// TIA Portal project "FactoryIO_Template" (V17)

(* hardware
DEVICE "S71500/ET200MP-Station_1"  S7-1500 station
   slot 0: "Profilschiene_0"  6ES7 590-1***0-0AA0
   slot 1: "PLC_1"  CPU 1511-1 PN  6ES7 511-1AK00-0AB0  V1.8
   slot 2: "AI 8xU/I/RTD/TC ST_1"  AI 8xU/I/RTD/TC ST  6ES7 531-7KF00-0AB0  V2.0
   slot 3: "AI 8xU/I/RTD/TC ST_2"  AI 8xU/I/RTD/TC ST  6ES7 531-7KF00-0AB0  V2.0
   slot 4: "AI 8xU/I/RTD/TC ST_3"  AI 8xU/I/RTD/TC ST  6ES7 531-7KF00-0AB0  V2.0
   slot 5: "AI 8xU/I/RTD/TC ST_4"  AI 8xU/I/RTD/TC ST  6ES7 531-7KF00-0AB0  V2.0
   slot 6: "DI 16x24VDC BA_1"  DI 16x24VDC BA  6ES7 521-1BH10-0AA0  V1.0
DEVICE "HMI_1"  TP700 Comfort
   slot 0: "HMI_1"  TP700 Comfort  6AV2 124-0GC01-0AX0  17.0.0.0
   slot 1: "HMI_RT_1"  TP700 Comfort  6AV2 124-0GC01-0AX0  17.0.0.0
   slot 5: "HMI_1.IE_CP_1"  PROFINET Interface  17.0.0.0
      slot 1: "PROFINET Interface_1"  PROFINET Interface
         slot 1: "Port_1"  Port
         slot 2: "Port_2"  Port
   slot 7: "HMI_1.MPI/DP_CP_1"  MPI/DP Interface  17.0.0.0
*)

// ===== PLC "PLC_1"  CPU 1511-1 PN =====

VAR_GLOBAL   // PLC tag table "Standard-Variablentabelle"
   "S" AT %E0.0 : Bool;   // capteur de présence du flacon sur le convoyeur 1
   "S21" AT %I0.7 : Bool;   // Convoyeur1
   "FCY" AT %I0.1 : Bool;   // arret urgence
   "DCY" AT %I0.3 : Bool;   // ok button
   "Me_1" AT %M0.0 : Bool;
   "EV" AT %Q0.1 : Bool;
   "S2" AT %I0.2 : Bool;
   "C2" AT %Q0.2 : Bool;
   "Me_2" AT %M0.1 : Bool;
   "C1" AT %Q0.0 : Bool;
   "movingX" AT %I0.5 : Bool;
   "movingZ" AT %I0.6 : Bool;
   "detected" AT %I0.4 : Bool;
   "pickZ" AT %Q0.3 : Bool;
   "pickX" AT %Q0.4 : Bool;
   "grab" AT %Q0.5 : Bool;
   "Tag_1" AT %M0.2 : Bool;
   "Tag_2" AT %M0.3 : Bool;
   "Tag_3" AT %M0.4 : Bool;
   "Tag_4" AT %M0.5 : Bool;
   "Tag_5" AT %M0.7 : Bool;
   "Tag_6" AT %M1.0 : Bool;
   "Tag_7" AT %M1.1 : Bool;
   "sd" AT %I1.0 : Bool;
   "cb" AT %Q0.6 : Bool;
   "Tag_8" AT %M1.2 : Bool;
   "Tag_9" AT %M1.3 : Bool;
   "Tag_10" AT %M1.4 : Bool;
   "Tag_11" AT %M1.5 : Bool;
   "C3" AT %Q0.7 : Bool;
   "AU" AT %I1.1 : Bool;
   "C4" AT %Q1.0 : Bool;
   "C6" AT %Q1.2 : Bool;
   "S3" AT %I1.2 : Bool;
   "C5" AT %Q1.1 : Bool;
   "S45" AT %I1.3 : Bool;
   "S5" AT %I1.4 : Bool;
   "Tag_12" AT %M1.6 : Bool;
   "C7" AT %Q1.3 : Bool;
   "S6" AT %I1.5 : Bool;
   "Tag_14" AT %M1.7 : Bool;
   "Tag_13" AT %M2.0 : Bool;
   "Tag_15" AT %M2.1 : Bool;
   "X" AT %QD30 : Real;
   "Z" AT %QD34 : Real;
   "Tag_16" AT %I1.6 : Bool;
   "Tag_17" AT %M2.2 : Bool;
   "Tag_18" AT %Q1.4 : Bool;
   "ZP" AT %ID30 : Real;
   "Tag_19" AT %M2.3 : Bool;
   "SensorZ" AT %I1.7 : Bool;
   "Tag_21" AT %M2.4 : Bool;
   "Tag_20" AT %Q1.5 : Bool;
   "Tag_22" AT %I2.1 : Bool;
   "Tag_23" AT %I2.0 : Bool;
   "Tag_24" AT %M2.5 : Bool;
   "start" AT %I2.2 : Bool;
   "Tag_26" AT %M2.6 : Bool;
   "Tag_27" AT %M2.7 : Bool;
   "C8" AT %Q1.6 : Bool;
   "Tag_30" AT %Q1.7 : Bool;
   "Tag_32" AT %M3.0 : Bool;
   "full" AT %I2.6 : Bool;
   "Tag_33" AT %M3.1 : Bool;
   "low" AT %I2.7 : Bool;
   "Tag_35" AT %Q2.5 : Bool;
   "Tag_36" AT %M3.2 : Bool;
   "discharge" AT %Q2.6 : Bool;
   "SS" AT %I2.3 : Bool;
   "startIHM" AT %I2.4 : Bool;
   "Tag_25" AT %M3.3 : Bool;
   "Tag_28" AT %M3.4 : Bool;
   "Tag_29" AT %M3.5 : Bool;
   "Tag_31" AT %I2.5 : Bool;
   "Tag_34" AT %M3.6 : Bool;
   "Tag_37" AT %MW4 : Int;
   "Tag_38" AT %M4.0 : Bool;
   "cv" AT %MW6 : Int;
   "Tag_39" AT %M4.1 : Bool;
END_VAR

// folder: System blocks/Program resources

DATA_BLOCK "T1"   // DB1
{ S7_Optimized_Access := 'TRUE' }
AUTHOR : Simatic
FAMILY : IEC
NAME : IEC_TMR
VERSION : 1.0
// stored: InstanceOfName IEC_TIMER
"IEC_TIMER"
BEGIN
END_DATA_BLOCK

DATA_BLOCK "T2"   // DB2
{ S7_Optimized_Access := 'TRUE' }
AUTHOR : Simatic
FAMILY : IEC
NAME : IEC_TMR
VERSION : 1.0
// stored: InstanceOfName IEC_TIMER
"IEC_TIMER"
BEGIN
END_DATA_BLOCK

DATA_BLOCK "T3"   // DB3
{ S7_Optimized_Access := 'TRUE' }
AUTHOR : Simatic
FAMILY : IEC
NAME : IEC_TMR
VERSION : 1.0
// stored: InstanceOfName IEC_TIMER
"IEC_TIMER"
BEGIN
END_DATA_BLOCK

DATA_BLOCK "T4"   // DB4
{ S7_Optimized_Access := 'TRUE' }
AUTHOR : Simatic
FAMILY : IEC
NAME : IEC_TMR
VERSION : 1.0
// stored: InstanceOfName IEC_TIMER
"IEC_TIMER"
BEGIN
END_DATA_BLOCK

DATA_BLOCK "com1"   // DB5
{ S7_Optimized_Access := 'TRUE' }
AUTHOR : Simatic
FAMILY : IEC
NAME : CNTR
VERSION : 1.0
// stored: InstanceOfName IEC_COUNTER
"IEC_COUNTER"
BEGIN
END_DATA_BLOCK

// folder: (top level)

FUNCTION "MHJ-PLC-Lab-Function-S71500" : Void   // FC9000, SCL
{ S7_Optimized_Access := 'TRUE' }
VERSION : 0.1
   VAR_TEMP
      Value : Byte;
      ForCounter : Int;
   END_VAR
   VAR CONSTANT
      Value_01_DW : DWord := 16#1223_5486;
      Value_02_DW : DWord := 16#A6C9_D1F5;
   END_VAR
BEGIN

   #Value:=PEEK(area := 16#82,
        dbNumber := 0,
        byteOffset := 511);
   #Value := #Value + 1;

   POKE(area := 16#82,
        dbNumber := 0,
        byteOffset := 511,
        value := #Value);

   POKE(area := 16#82,
        dbNumber := 0,
        byteOffset := 1016,
        value := #Value_01_DW);
   POKE(area := 16#82,
        dbNumber := 0,
        byteOffset := 1020,
        value := #Value_02_DW);

   FOR #ForCounter := 0 TO 63 DO
       #Value:=PEEK(area := 16#1,
            dbNumber := 0,
            byteOffset := #ForCounter);
       POKE(area := 16#81,
            dbNumber := 0,
            byteOffset := #ForCounter,
            value := #Value);
   END_FOR;
   #Value := PEEK(area := 16#1,
                  dbNumber := 0,
                  byteOffset := 512);
   POKE(area := 16#82,
        dbNumber := 0,
        byteOffset := 512,
        value := #Value);
END_FUNCTION

ORGANIZATION_BLOCK "Main"   // OB1, LAD, ProgramCycle
TITLE = "Main Program Sweep (Cycle)"
{ S7_Optimized_Access := 'TRUE' }
VERSION : 0.1
   VAR_INPUT
      Initial_Call : Bool;   // Initial call of this OB
      Remanence : Bool;   // =True, if remanent data are available
   END_VAR
   VAR_TEMP   // added for the SCL form of the ladder/FBD networks
      _w1 : Bool;
      _w2 : Bool;
   END_VAR
BEGIN

REGION Network 1
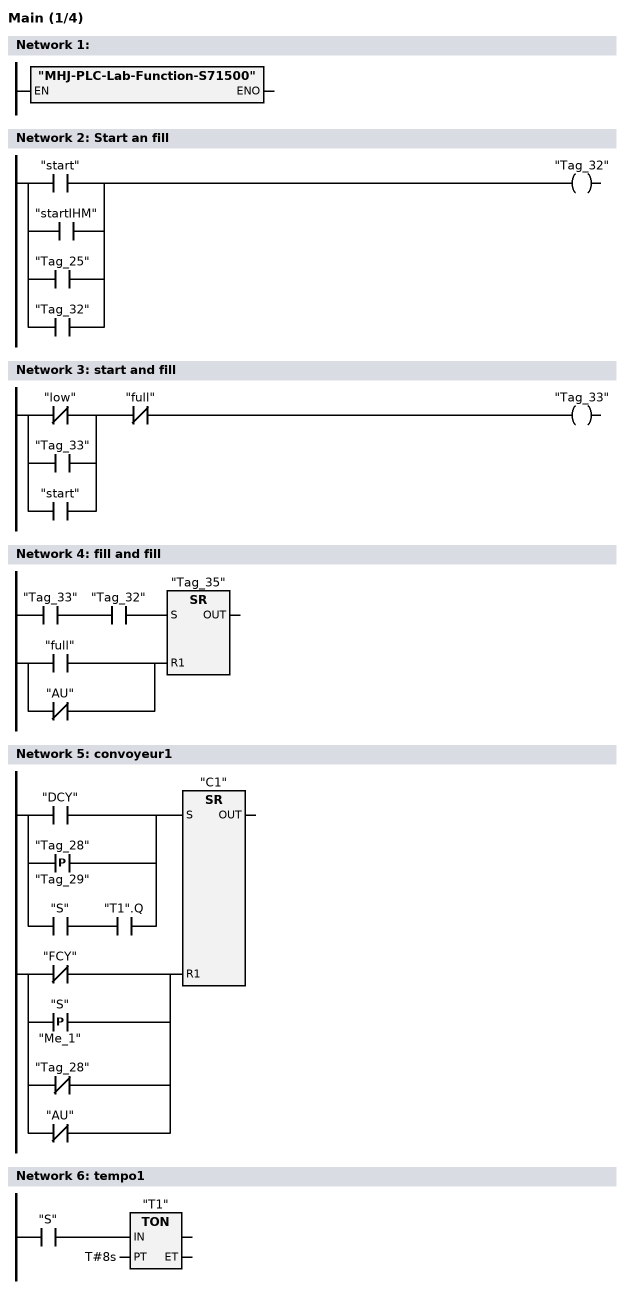
   RUNG wire#powerrail
      "MHJ-PLC-Lab-Function-S71500"()
   END_RUNG
   // the same network as SCL:
   "MHJ-PLC-Lab-Function-S71500"();
END_REGION

REGION Network 2: Start an fill
   RUNG wire#powerrail
      Contact( "start" )
      wire#w1
      Coil( "Tag_32" )
   END_RUNG
   RUNG wire#powerrail
      Contact( "startIHM" )
   END_RUNG wire#w1
   RUNG wire#powerrail
      Contact( "Tag_25" )
   END_RUNG wire#w1
   RUNG wire#powerrail
      Contact( "Tag_32" )
   END_RUNG wire#w1
   // the same network as SCL:
   "Tag_32" := "start" OR "startIHM" OR "Tag_25" OR "Tag_32";
END_REGION

REGION Network 3: start and fill
   RUNG wire#powerrail
      I_Contact( "low" )
      wire#w1
      I_Contact( "full" )
      Coil( "Tag_33" )
   END_RUNG
   RUNG wire#powerrail
      Contact( "Tag_33" )
   END_RUNG wire#w1
   RUNG wire#powerrail
      Contact( "start" )
   END_RUNG wire#w1
   // the same network as SCL:
   "Tag_33" := (NOT "low" OR "Tag_33" OR "start") AND NOT "full";
END_REGION

REGION Network 4: fill and fill
   RUNG wire#powerrail
      Contact( "Tag_33" )
      Contact( "Tag_32" )
      S_SR(operand := "Tag_35", r1 := wire#w1)
   END_RUNG
   RUNG wire#powerrail
      Contact( "full" )
   END_RUNG wire#w1
   RUNG wire#powerrail
      I_Contact( "AU" )
   END_RUNG wire#w1
   // the same network as SCL:
   IF "Tag_33" AND "Tag_32" THEN
       "Tag_35" := TRUE;   // SR flip-flop
   END_IF;
   IF "full" OR NOT "AU" THEN "Tag_35" := FALSE; END_IF;
END_REGION

REGION Network 5: convoyeur1
   RUNG wire#powerrail
      Contact( "DCY" )
      wire#w1
      S_SR(operand := "C1", r1 := wire#w2)
   END_RUNG
   RUNG wire#powerrail
      P_Contact(operand := "Tag_28", bit := "Tag_29")
   END_RUNG wire#w1
   RUNG wire#powerrail
      Contact( "S" )
      Contact( "T1".Q )
   END_RUNG wire#w1
   RUNG wire#powerrail
      I_Contact( "FCY" )
   END_RUNG wire#w2
   RUNG wire#powerrail
      P_Contact(operand := "S", bit := "Me_1")
   END_RUNG wire#w2
   RUNG wire#powerrail
      I_Contact( "Tag_28" )
   END_RUNG wire#w2
   RUNG wire#powerrail
      I_Contact( "AU" )
   END_RUNG wire#w2
   // the same network as SCL:
   #_w1 := "Tag_28" AND NOT "Tag_29";   // rising edge of "Tag_28"
   "Tag_29" := "Tag_28";
   #_w2 := "S" AND NOT "Me_1";   // rising edge of "S"
   "Me_1" := "S";
   IF "DCY" OR #_w1 OR ("S" AND "T1".Q) THEN
       "C1" := TRUE;   // SR flip-flop
   END_IF;
   IF NOT "FCY" OR #_w2 OR NOT "Tag_28" OR NOT "AU" THEN "C1" := FALSE; END_IF;
END_REGION

REGION Network 6: tempo1
   "T1".TON(IN := "S", PT := T#8s);
END_REGION

REGION Network 7: electrovanne
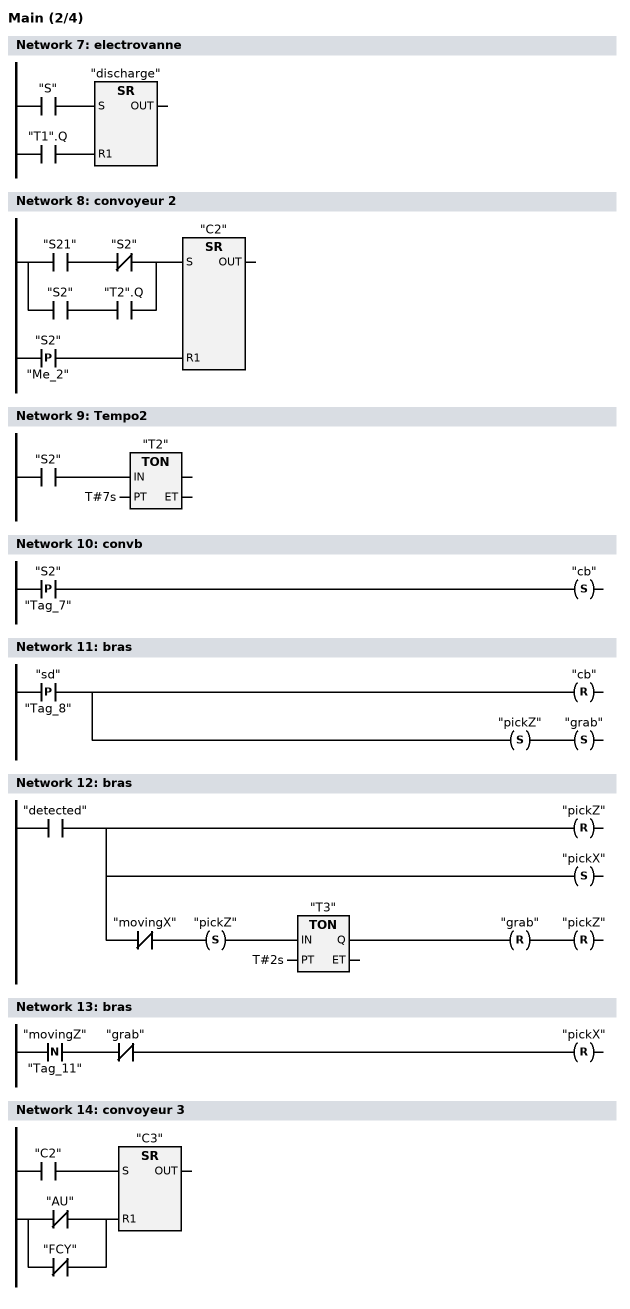
   RUNG wire#powerrail
      Contact( "S" )
      S_SR(operand := "discharge", r1 := wire#w1)
   END_RUNG
   RUNG wire#powerrail
      Contact( "T1".Q )
   END_RUNG wire#w1
   // the same network as SCL:
   IF "S" THEN
       "discharge" := TRUE;   // SR flip-flop
   END_IF;
   IF "T1".Q THEN "discharge" := FALSE; END_IF;
END_REGION

REGION Network 8: convoyeur 2
   RUNG wire#powerrail
      Contact( "S21" )
      I_Contact( "S2" )
      wire#w1
      S_SR(operand := "C2", r1 := wire#w2)
   END_RUNG
   RUNG wire#powerrail
      Contact( "S2" )
      Contact( "T2".Q )
   END_RUNG wire#w1
   RUNG wire#powerrail
      P_Contact(operand := "S2", bit := "Me_2")
   END_RUNG wire#w2
   // the same network as SCL:
   #_w1 := "S2" AND NOT "Me_2";   // rising edge of "S2"
   "Me_2" := "S2";
   IF ("S21" AND NOT "S2") OR ("S2" AND "T2".Q) THEN
       "C2" := TRUE;   // SR flip-flop
   END_IF;
   IF #_w1 THEN "C2" := FALSE; END_IF;
END_REGION

REGION Network 9: Tempo2
   "T2".TON(IN := "S2", PT := T#7s);
END_REGION

REGION Network 10: convb
   RUNG wire#powerrail
      P_Contact(operand := "S2", bit := "Tag_7")
      S_Coil( "cb" )
   END_RUNG
   // the same network as SCL:
   #_w1 := "S2" AND NOT "Tag_7";   // rising edge of "S2"
   "Tag_7" := "S2";
   IF #_w1 THEN "cb" := TRUE; END_IF;
END_REGION

REGION Network 11: bras
   RUNG wire#powerrail
      P_Contact(operand := "sd", bit := "Tag_8")
      wire#w1
      R_Coil( "cb" )
   END_RUNG
   RUNG wire#w1
      S_Coil( "pickZ" )
      S_Coil( "grab" )
   END_RUNG
   // the same network as SCL:
   #_w1 := "sd" AND NOT "Tag_8";   // rising edge of "sd"
   "Tag_8" := "sd";
   IF #_w1 THEN
       "cb" := FALSE;
       "pickZ" := TRUE;
       "grab" := TRUE;
   END_IF;
END_REGION

REGION Network 12: bras
   IF "detected" THEN
       "pickZ" := FALSE;
       "pickX" := TRUE;
   END_IF;
   #_w1 := "detected" AND NOT "movingX";
   IF #_w1 THEN "pickZ" := TRUE; END_IF;
   "T3".TON(IN := #_w1, PT := T#2s);
   IF "T3".Q THEN
       "grab" := FALSE;
       "pickZ" := FALSE;
   END_IF;
END_REGION

REGION Network 13: bras
   RUNG wire#powerrail
      N_Contact(operand := "movingZ", bit := "Tag_11")
      I_Contact( "grab" )
      R_Coil( "pickX" )
   END_RUNG
   // the same network as SCL:
   #_w1 := NOT "movingZ" AND "Tag_11";   // falling edge of "movingZ"
   "Tag_11" := "movingZ";
   IF #_w1 AND NOT "grab" THEN "pickX" := FALSE; END_IF;
END_REGION

REGION Network 14: convoyeur 3
   RUNG wire#powerrail
      Contact( "C2" )
      S_SR(operand := "C3", r1 := wire#w1)
   END_RUNG
   RUNG wire#powerrail
      I_Contact( "AU" )
   END_RUNG wire#w1
   RUNG wire#powerrail
      I_Contact( "FCY" )
   END_RUNG wire#w1
   // the same network as SCL:
   IF "C2" THEN
       "C3" := TRUE;   // SR flip-flop
   END_IF;
   IF NOT "AU" OR NOT "FCY" THEN "C3" := FALSE; END_IF;
END_REGION

REGION Network 15: convoyeur 4
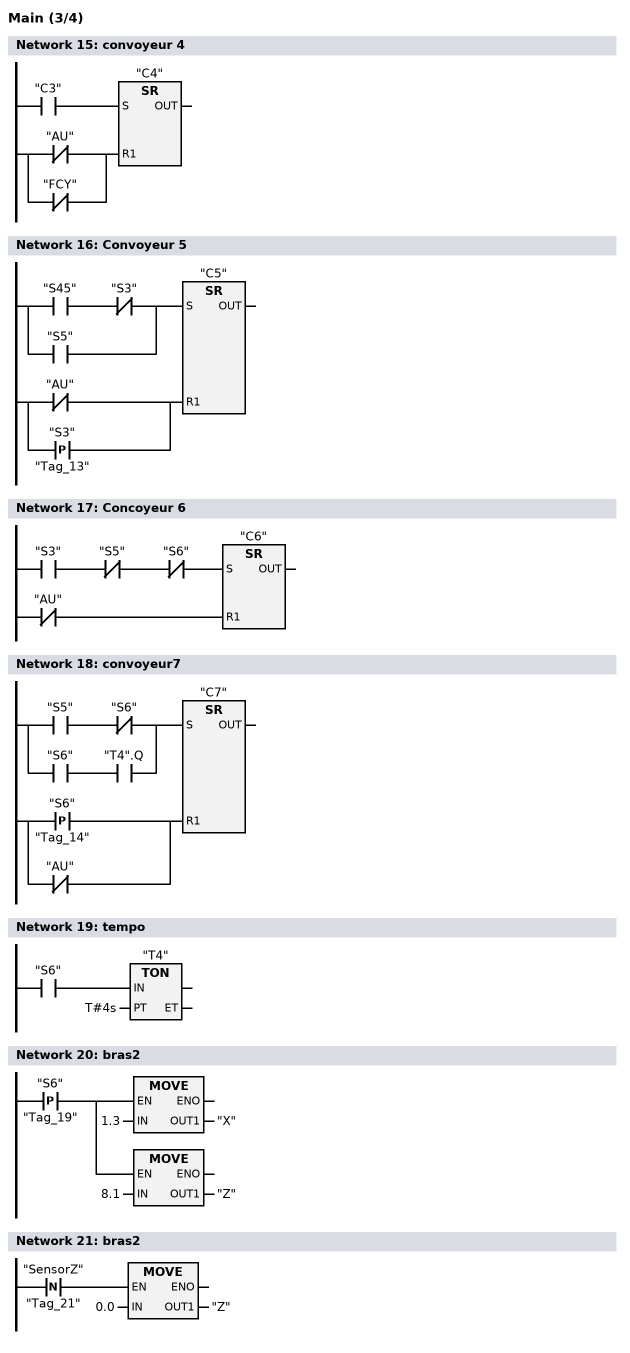
   RUNG wire#powerrail
      Contact( "C3" )
      S_SR(operand := "C4", r1 := wire#w1)
   END_RUNG
   RUNG wire#powerrail
      I_Contact( "AU" )
   END_RUNG wire#w1
   RUNG wire#powerrail
      I_Contact( "FCY" )
   END_RUNG wire#w1
   // the same network as SCL:
   IF "C3" THEN
       "C4" := TRUE;   // SR flip-flop
   END_IF;
   IF NOT "AU" OR NOT "FCY" THEN "C4" := FALSE; END_IF;
END_REGION

REGION Network 16: Convoyeur 5
   RUNG wire#powerrail
      Contact( "S45" )
      I_Contact( "S3" )
      wire#w1
      S_SR(operand := "C5", r1 := wire#w2)
   END_RUNG
   RUNG wire#powerrail
      Contact( "S5" )
   END_RUNG wire#w1
   RUNG wire#powerrail
      I_Contact( "AU" )
   END_RUNG wire#w2
   RUNG wire#powerrail
      P_Contact(operand := "S3", bit := "Tag_13")
   END_RUNG wire#w2
   // the same network as SCL:
   #_w1 := "S3" AND NOT "Tag_13";   // rising edge of "S3"
   "Tag_13" := "S3";
   IF ("S45" AND NOT "S3") OR "S5" THEN
       "C5" := TRUE;   // SR flip-flop
   END_IF;
   IF NOT "AU" OR #_w1 THEN "C5" := FALSE; END_IF;
END_REGION

REGION Network 17: Concoyeur 6
   RUNG wire#powerrail
      Contact( "S3" )
      I_Contact( "S5" )
      I_Contact( "S6" )
      S_SR(operand := "C6", r1 := wire#w1)
   END_RUNG
   RUNG wire#powerrail
      I_Contact( "AU" )
   END_RUNG wire#w1
   // the same network as SCL:
   IF "S3" AND NOT "S5" AND NOT "S6" THEN
       "C6" := TRUE;   // SR flip-flop
   END_IF;
   IF NOT "AU" THEN "C6" := FALSE; END_IF;
END_REGION

REGION Network 18: convoyeur7
   RUNG wire#powerrail
      Contact( "S5" )
      I_Contact( "S6" )
      wire#w1
      S_SR(operand := "C7", r1 := wire#w2)
   END_RUNG
   RUNG wire#powerrail
      Contact( "S6" )
      Contact( "T4".Q )
   END_RUNG wire#w1
   RUNG wire#powerrail
      P_Contact(operand := "S6", bit := "Tag_14")
   END_RUNG wire#w2
   RUNG wire#powerrail
      I_Contact( "AU" )
   END_RUNG wire#w2
   // the same network as SCL:
   #_w1 := "S6" AND NOT "Tag_14";   // rising edge of "S6"
   "Tag_14" := "S6";
   IF ("S5" AND NOT "S6") OR ("S6" AND "T4".Q) THEN
       "C7" := TRUE;   // SR flip-flop
   END_IF;
   IF #_w1 OR NOT "AU" THEN "C7" := FALSE; END_IF;
END_REGION

REGION Network 19: tempo
   "T4".TON(IN := "S6", PT := T#4s);
END_REGION

REGION Network 20: bras2
   RUNG wire#powerrail
      P_Contact(operand := "S6", bit := "Tag_19")
      wire#w1
      Move(in := 1.3, out1 => "X")
   END_RUNG
   RUNG wire#w1
      Move(in := 8.1, out1 => "Z")
   END_RUNG
   // the same network as SCL:
   #_w1 := "S6" AND NOT "Tag_19";   // rising edge of "S6"
   "Tag_19" := "S6";
   IF #_w1 THEN
       "X" := 1.3;
       "Z" := 8.1;
   END_IF;
END_REGION

REGION Network 21: bras2
   RUNG wire#powerrail
      N_Contact(operand := "SensorZ", bit := "Tag_21")
      Move(in := 0.0, out1 => "Z")
   END_RUNG
   // the same network as SCL:
   #_w1 := NOT "SensorZ" AND "Tag_21";   // falling edge of "SensorZ"
   "Tag_21" := "SensorZ";
   IF #_w1 THEN "Z" := 0.0; END_IF;
END_REGION

REGION Network 22: Classification
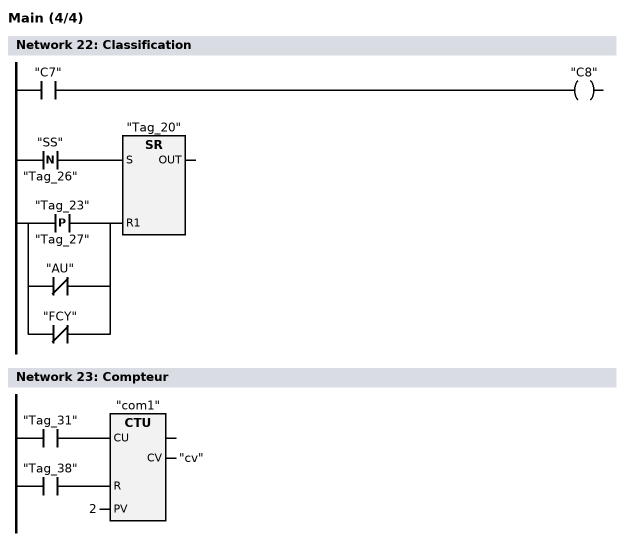
   RUNG wire#powerrail
      Contact( "C7" )
      Coil( "C8" )
   END_RUNG
   RUNG wire#powerrail
      N_Contact(operand := "SS", bit := "Tag_26")
      S_SR(operand := "Tag_20", r1 := wire#w1)
   END_RUNG
   RUNG wire#powerrail
      P_Contact(operand := "Tag_23", bit := "Tag_27")
   END_RUNG wire#w1
   RUNG wire#powerrail
      I_Contact( "AU" )
   END_RUNG wire#w1
   RUNG wire#powerrail
      I_Contact( "FCY" )
   END_RUNG wire#w1
   // the same network as SCL:
   "C8" := "C7";
   #_w1 := NOT "SS" AND "Tag_26";   // falling edge of "SS"
   "Tag_26" := "SS";
   #_w2 := "Tag_23" AND NOT "Tag_27";   // rising edge of "Tag_23"
   "Tag_27" := "Tag_23";
   IF #_w1 THEN
       "Tag_20" := TRUE;   // SR flip-flop
   END_IF;
   IF #_w2 OR NOT "AU" OR NOT "FCY" THEN "Tag_20" := FALSE; END_IF;
END_REGION

REGION Network 23: Compteur
   "com1".CTU(CU := "Tag_31", R := "Tag_38", PV := 2, CV => "cv");
END_REGION
END_ORGANIZATION_BLOCK

(* ===== HMI "HMI_RT_1" =====
system functions are stored by id; their names below are inferred from use
connection "HMI_Connection_1": ETHERNET, S7_1500_OMS

HMI tags "Default tag table"
   "start" : Bool = PLC startIHM AT %I2.4, 1 s
   "AU" : Bool = PLC AU AT %I1.1, 1 s
   "FCY" : Bool = PLC FCY AT %I0.1, 1 s
   "Tag_25" : Bool = PLC Tag_25 AT %M3.3, 1 s
   "Tag_28" : Bool = PLC Tag_28 AT %M3.4, 1 s
   "cv" : Int = PLC cv AT %MW6, 1 s
   "Tag_38" : Bool = PLC Tag_38 AT %M4.0, 1 s

screen "Root screen" 800x420, template "Template_1"
   Button "Button_2" at 291,114 size 132x32; TextOff 'Début cycle'
      on Click: SetBit("Tag_28")
   Button "Button_3" at 527,115 size 96x32; TextOff 'Fin cycle'
      on Click: SetBit("FCY")
   Button "Button_4" at 425,289 size 194x32; TextOff 'Emergency Stop'
      on Click: SetBit("AU")
   Button "Button_5" at 91,114 size 96x32; TextOff 'Start'
      on Click: SetBit("Tag_25")
   IOField "I/O field_2" at 49,289 size 96x32; FormatPattern 999
      ProcessValue <- "cv"
      on Deactivate: ResetBit(N)
   Button "Button_1" at 40,238 size 253x32; TextOff 'Compteur des flacons'
   Button "Button_6" at 192,289 size 96x32; TextOff 'RESET'
      on Click: SetBit("Tag_38")

Template "Template_1" 800x420
   Button "Exit" at 720,360 size 78x58; TextOff 'Exit'; PictureOff "ExitRuntime_TP700_Comfort_TR"; PictureOn "ExitRuntime_TP700_Comfort_TR"
      on Release: StopRuntime(0)
   Button "Template_Button" at 640,360 size 78x58; TextOff 'Text'
   Button "Template_Button_1" at 560,360 size 78x58; TextOff 'Text'
   Button "Template_Button_2" at 480,360 size 78x58; TextOff 'Text'
   Button "Template_Button_3" at 400,360 size 78x58; TextOff 'Text'
   Button "Template_Button_4" at 321,360 size 78x58; TextOff 'Text'
   Button "Template_Button_5" at 241,360 size 78x58; TextOff 'Text'
   Button "Template_Button_6" at 161,360 size 78x58; TextOff 'Text'
   Button "Alarms" at 81,360 size 78x58; TextOff 'Alarms'; PictureOff "AlarmDisplay_TP700_Comfort_TR"; PictureOn "AlarmDisplay_TP700_Comfort_TR"
      on Release: function_ef3f5d25("Alarm window_Unacknowledged", -1)
   Button "Start screen" at 1,360 size 78x58; TextOff 'Start screen'; PictureOff "NavigateHome_TP700_Comfort_TR"; PictureOn "NavigateHome_TP700_Comfort_TR"
      on Release: ActivateScreen("Root screen", 0)
*)